ABB RAPID module: P2540SegmentOrg.mod

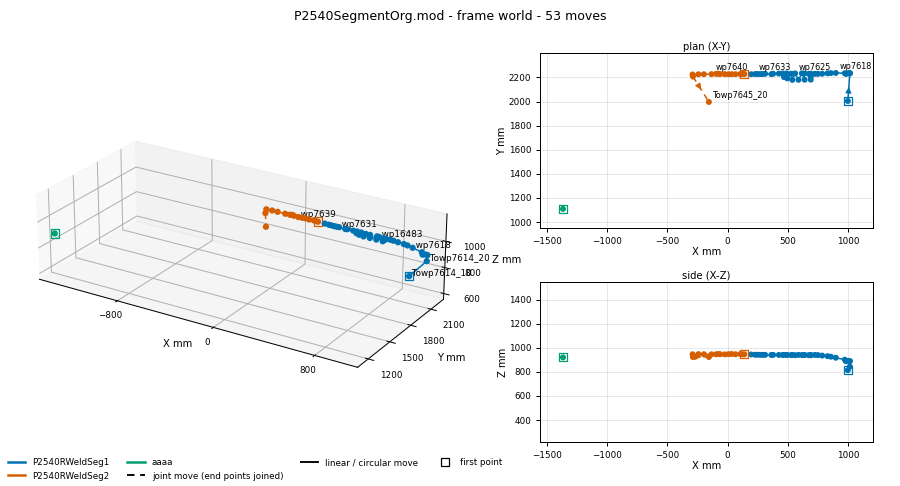
[picture p0: tool path of P2540SegmentOrg.mod in frame world, 53 of 55 moves have a stored position in this frame; points joined in program order, loops and branches not executed]
%%%
   VERSION: 1
   LANGUAGE: ENGLISH
%%%

MODULE P2540Segment
  !********************************
  !*                              *
  !*   Module : P2540Segment.mod   *
  !*   Name   : R1 =2V2=V3AR22    *
  !*   Robot  : 66-60648          *
  !*   Task   : T_Rob1            *
  !*   Vers.  : 7.3               *
  !*                              *
  !********************************
  !
  !
  !============================
  ! Jointtarget for - P2540  -
  !============================
  ! jointtarget for start and stop schedule
  LOCAL CONST jointtarget StartSchedule:=[[23.5621,-44.1357,51.2586,26.8219,73.3194,-96.4131],[9E+09,30.0007,9E+09,9E+09,9E+09,9E+09]];
  LOCAL CONST jointtarget EndSchedule:=[[23.5621,-44.1357,51.2586,26.8219,73.3194,-96.4131],[9E+09,30.0007,9E+09,9E+09,9E+09,9E+09]];
  !
  !
  !===========
  ! Robtarget
  !===========
  ! robtarget for P2540  Right
  LOCAL CONST robtarget Towp7614_10:=[[2081.47,305.36,1121.56],[0.00371606,0.598737,0.800932,-0.000148476],[0,0,-1,0],[9E+09,79.9999,9E+09,9E+09,9E+09,9E+09]];
  LOCAL CONST robtarget Towp7614_20:=[[2062.30,533.66,1090.73],[0.0314135,-0.610941,-0.788905,0.0581832],[0,0,-1,0],[9E+09,59.9996,9E+09,9E+09,9E+09,9E+09]];
  LOCAL CONST robtarget wp7614:=[[2060.79,536.44,1045.07],[0.0756945,-0.590813,-0.799762,0.0747174],[0,0,-1,0],[9E+09,27.201,9E+09,9E+09,9E+09,9E+09]];
  LOCAL CONST robtarget wp7615:=[[2072.79,535.23,1043.37],[0.0761961,-0.650595,-0.752147,0.0720186],[0,0,-1,0],[9E+09,21.5173,9E+09,9E+09,9E+09,9E+09]];
  LOCAL CONST robtarget wp7616:=[[2104.65,535.90,1033.71],[0.0596176,-0.670701,-0.735912,0.0709296],[0,0,-1,0],[9E+09,20.2489,9E+09,9E+09,9E+09,9E+09]];
  LOCAL CONST robtarget wp7619:=[[2219.57,538.20,1009.48],[0.0741953,-0.671905,-0.735684,0.0424222],[0,0,-1,0],[9E+09,27.2002,9E+09,9E+09,9E+09,9E+09]];
  LOCAL CONST robtarget wp7620:=[[2247.39,536.95,1005.37],[0.0595264,-0.701649,-0.708305,0.0494151],[0,0,-1,0],[9E+09,27.2002,9E+09,9E+09,9E+09,9E+09]];
  LOCAL CONST robtarget wp7621:=[[2292.13,533.79,1000.70],[0.0332252,-0.730819,-0.681624,0.013398],[0,0,-1,0],[9E+09,28.1993,9E+09,9E+09,9E+09,9E+09]];
  LOCAL CONST robtarget wp7622:=[[2327.33,533.09,996.92],[0.0333113,-0.730834,-0.681602,0.0134842],[0,0,-1,0],[9E+09,27.2006,9E+09,9E+09,9E+09,9E+09]];
  LOCAL CONST robtarget wp7623:=[[2353.30,533.71,995.86],[0.0293606,-0.749439,-0.661259,0.0143902],[0,0,-1,0],[9E+09,27.1999,9E+09,9E+09,9E+09,9E+09]];
  LOCAL CONST robtarget wp16388:=[[2387.90,486.12,997.86],[0.00612508,-0.760122,-0.649737,-0.00322363],[0,0,-1,0],[9E+09,4.11012,9E+09,9E+09,9E+09,9E+09]];
  LOCAL CONST robtarget wp22643:=[[2386.96,534.93,997.70],[0.0127164,-0.751544,-0.659552,0.00163492],[0,0,-1,0],[9E+09,29.9002,9E+09,9E+09,9E+09,9E+09]];
  LOCAL CONST robtarget wp7624:=[[2405.02,534.99,998.03],[0.000354615,0.772557,0.634784,0.0140377],[0,0,-1,0],[9E+09,29.8997,9E+09,9E+09,9E+09,9E+09]];
  LOCAL CONST robtarget wp16483:=[[2442.71,537.01,996.52],[0.0171293,-0.772749,-0.634461,-0.00402584],[0,0,-1,0],[9E+09,29.9002,9E+09,9E+09,9E+09,9E+09]];
  LOCAL CONST robtarget wp16482:=[[2480.83,537.98,1000.06],[0.000439903,0.773189,0.634169,-0.000630514],[0,0,-1,0],[9E+09,32.3991,9E+09,9E+09,9E+09,9E+09]];
  LOCAL CONST robtarget wp16389:=[[2438.79,486.06,996.71],[0.00848171,-0.773071,-0.634066,-0.0155309],[0,0,-1,0],[9E+09,27.1999,9E+09,9E+09,9E+09,9E+09]];
  LOCAL CONST robtarget wp16390:=[[2489.71,485.99,996.41],[0.0138037,-0.776796,-0.629424,-0.0146608],[0,0,-1,0],[9E+09,4.07069,9E+09,9E+09,9E+09,9E+09]];
  LOCAL CONST robtarget wp7625:=[[2516.82,539.27,998.69],[0.0143354,-0.773193,-0.633743,-0.0181102],[0,0,-1,0],[9E+09,40.9991,9E+09,9E+09,9E+09,9E+09]];
  LOCAL CONST robtarget wp16391:=[[2540.52,486.02,996.53],[0.0108996,-0.789577,-0.613522,-0.00567082],[0,0,-1,0],[9E+09,4.11961,9E+09,9E+09,9E+09,9E+09]];
  LOCAL CONST robtarget wp7626:=[[2549.80,537.47,998.38],[0.00989104,-0.789531,-0.61347,-0.0137525],[0,0,-1,0],[9E+09,32.3999,9E+09,9E+09,9E+09,9E+09]];
  LOCAL CONST robtarget wp16392:=[[2582.12,498.78,997.71],[0.00612506,-0.789608,-0.613429,-0.0133152],[0,0,-1,0],[9E+09,27.3998,9E+09,9E+09,9E+09,9E+09]];
  LOCAL CONST robtarget wp7628:=[[2620.20,540.35,997.67],[0.00660724,0.789817,0.61328,0.00488902],[0,0,-1,0],[9E+09,32.3997,9E+09,9E+09,9E+09,9E+09]];
  LOCAL CONST robtarget wp7630:=[[2652.05,539.44,997.26],[0.00765265,-0.811596,-0.584132,-0.00589266],[0,0,-1,0],[9E+09,32.4003,9E+09,9E+09,9E+09,9E+09]];


  LOCAL CONST robtarget wp16473:=[[2699.16,538.68,997.15],[0.00502678,-0.811529,-0.584197,-0.0100621],[0,0,-1,0],[9E+09,29.9001,9E+09,9E+09,9E+09,9E+09]];
  LOCAL CONST robtarget wp16471:=[[2713.62,536.00,997.85],[0.0220624,-0.810911,-0.584577,-0.0140417],[0,0,-1,0],[9E+09,29.8894,9E+09,9E+09,9E+09,9E+09]];
  LOCAL CONST robtarget wp16472:=[[2727.21,534.57,998.78],[0.000173773,-0.813784,-0.58116,-0.000410488],[0,0,-1,0],[9E+09,31.0445,9E+09,9E+09,9E+09,9E+09]];
  LOCAL CONST robtarget wp7631:=[[2765.83,539.26,997.19],[0.00454817,-0.812585,-0.582806,0.0035711],[0,0,-1,0],[9E+09,29.9004,9E+09,9E+09,9E+09,9E+09]];
  LOCAL CONST robtarget wp31008:=[[2786.44,538.03,997.19],[0.00908552,-0.814655,-0.579848,0.00473351],[0,0,-1,0],[9E+09,29.9001,9E+09,9E+09,9E+09,9E+09]];

  LOCAL CONST robtarget wp7632:=[[2806.45,537.63,997.32],[0.00900133,0.815927,0.578044,0.00628094],[0,0,-1,0],[9E+09,30.0007,9E+09,9E+09,9E+09,9E+09]];
  LOCAL CONST robtarget wp31009:=[[2829.93,538.04,996.73],[0.00768568,0.812719,0.582397,0.0152683],[0,0,-1,0],[9E+09,29.9005,9E+09,9E+09,9E+09,9E+09]];

  LOCAL CONST robtarget wp7633:=[[2848.76,538.17,996.85],[0.00725543,0.810933,0.585076,0.00354437],[0,0,-1,0],[9E+09,29.8994,9E+09,9E+09,9E+09,9E+09]];
  LOCAL CONST robtarget wp7634:=[[2881.59,537.27,994.84],[0.0105951,-0.810906,-0.585073,-0.000189071],[0,0,-1,0],[9E+09,29.9002,9E+09,9E+09,9E+09,9E+09]];
  LOCAL CONST robtarget wp16150:=[[2938.22,539.11,993.71],[0.0155581,-0.812601,-0.582198,-0.0217884],[0,0,-1,0],[9E+09,29.9001,9E+09,9E+09,9E+09,9E+09]];
  LOCAL CONST robtarget wp16151:=[[2973.15,539.53,991.63],[0.0143352,-0.812577,-0.582323,-0.0201075],[0,0,-1,0],[9E+09,29.9001,9E+09,9E+09,9E+09,9E+09]];
  LOCAL CONST robtarget wp7636:=[[3012.11,539.12,993.74],[0.0076257,-0.811727,-0.583768,-0.0157572],[0,0,-1,0],[9E+09,27.2002,9E+09,9E+09,9E+09,9E+09]];
  LOCAL CONST robtarget wp7637:=[[3043.26,539.70,991.91],[0.0186046,-0.811439,-0.583534,-0.0264702],[0,0,-1,0],[9E+09,27.1997,9E+09,9E+09,9E+09,9E+09]];
  LOCAL CONST robtarget wp7638:=[[3070.27,539.54,992.95],[0.00847598,-0.813252,-0.581717,-0.0120917],[0,0,-1,0],[9E+09,27.2002,9E+09,9E+09,9E+09,9E+09]];
  LOCAL CONST robtarget wp7639:=[[3100.66,540.23,995.08],[0.00913472,-0.865282,-0.500928,-0.0163131],[0,0,-1,0],[9E+09,27.2002,9E+09,9E+09,9E+09,9E+09]];
  LOCAL CONST robtarget wp16146:=[[3138.44,541.78,994.19],[0.0055009,-0.894006,-0.447865,-0.0114338],[0,0,-1,0],[9E+09,29.9001,9E+09,9E+09,9E+09,9E+09]];
  LOCAL CONST robtarget wp16411:=[[3156.07,537.38,997.99],[0.00338754,0.895748,0.444538,0.00149798],[0,0,-1,0],[9E+09,60,9E+09,9E+09,9E+09,9E+09]];
  LOCAL CONST robtarget wp16147:=[[3173.12,543.64,994.77],[0.00345947,-0.894048,-0.447902,-0.00641748],[0,0,-1,0],[9E+09,29.9004,9E+09,9E+09,9E+09,9E+09]];
  LOCAL CONST robtarget wp7640:=[[3210.69,541.93,995.09],[0.00726479,-0.896754,-0.442203,-0.0150922],[0,0,-1,0],[9E+09,27.2006,9E+09,9E+09,9E+09,9E+09]];
  LOCAL CONST robtarget wp7642:=[[3274.35,542.16,994.69],[0.00655286,-0.899967,-0.435565,-0.0170478],[0,0,-1,0],[9E+09,27.1997,9E+09,9E+09,9E+09,9E+09]];
  LOCAL CONST robtarget wp7643:=[[3319.94,541.93,994.28],[0.00891136,-0.924508,-0.380439,-0.0215371],[0,0,-1,0],[9E+09,27.2002,9E+09,9E+09,9E+09,9E+09]];
  LOCAL CONST robtarget wp7644:=[[3368.35,541.38,995.77],[0.0101282,-0.928939,-0.369177,-0.0258691],[0,0,-1,0],[9E+09,27.1991,9E+09,9E+09,9E+09,9E+09]];
  LOCAL CONST robtarget Towp7645_20:=[[3235.39,311.48,1018.62],[0.00729107,-0.929368,-0.369063,0.00225485],[0,0,-2,0],[9E+09,58.7207,9E+09,9E+09,9E+09,9E+09]];
  LOCAL CONST robtarget Towp7645_30:=[[3678.48,197.21,1015.08],[0.00379367,0.692205,0.721685,0.000353803],[1,-1,0,0],[9E+09,50,9E+09,9E+09,9E+09,9E+09]];
  LOCAL CONST robtarget wp7645:=[[3426.32,542.43,994.99],[0.0229346,-0.426697,-0.903983,-0.014501],[1,-1,0,0],[9E+09,25,9E+09,9E+09,9E+09,9E+09]];
  LOCAL CONST robtarget wp7647:=[[3515.94,541.61,994.94],[0.0180354,-0.560505,-0.827819,-0.0147185],[1,-1,0,0],[9E+09,20,9E+09,9E+09,9E+09,9E+09]];
  LOCAL CONST robtarget wp7648:=[[3566.36,543.48,994.12],[0.000513143,0.675137,0.737686,-0.000593508],[1,-1,0,0],[9E+09,20,9E+09,9E+09,9E+09,9E+09]];
  LOCAL CONST robtarget wp7649:=[[3616.27,543.9,993.12],[0.000208783,0.783466,0.621428,-0.00029122],[1,0,-1,0],[9E+09,20,9E+09,9E+09,9E+09,9E+09]];

  LOCAL CONST robtarget Frwp6240_20:=[[3468.86,140.72,795.38],[0.00296039,0.761935,0.647638,0.001747],[1,-1,0,0],[9E+09,35.3553,9E+09,9E+09,9E+09,9E+09]];
  !
  !==========
  ! WobjData
  !==========
  ! wobj for spot welding P2540 Right
  PERS wobjdata wP2540_CabFrame:=[FALSE,TRUE,"",[[3089,1731.03,1926.23],[0.00267617,0.00632448,-0.999974,0.00237532]],[[0,0,0],[1,0,0,0]]];
  !
  !
  !==========
  ! SpotData
  !==========
  ! spot data P2540  Right
  LOCAL PERS spotdata Sd_wp7614_30:=[00761430,0,0,0,0];
  LOCAL PERS spotdata Sd_wp7615_30:=[00761530,0,0,0,0];
  LOCAL PERS spotdata Sd_wp7616_30:=[00761630,0,0,0,0];
  LOCAL PERS spotdata Sd_wp7619_30:=[00761930,0,0,0,0];
  LOCAL PERS spotdata Sd_wp7620_30:=[00762030,0,0,0,0];
  LOCAL PERS spotdata Sd_wp7621_30:=[00762130,0,0,0,0];
  LOCAL PERS spotdata Sd_wp7622_30:=[00762230,0,0,0,0];
  LOCAL PERS spotdata Sd_wp7623_30:=[00762330,0,0,0,0];
  LOCAL PERS spotdata Sd_wp7624_30:=[00762430,0,0,0,0];
  LOCAL PERS spotdata Sd_wp16483_30:=[01648330,0,0,0,0];
  LOCAL PERS spotdata Sd_wp16389_30:=[01638930,0,0,0,0];
  LOCAL PERS spotdata Sd_wp16482_30:=[01648230,0,0,0,0];
  LOCAL PERS spotdata Sd_wp16390_30:=[01639030,0,0,0,0];
  LOCAL PERS spotdata Sd_wp7625_30:=[00762530,0,0,0,0];
  LOCAL PERS spotdata Sd_wp16391_30:=[01639130,0,0,0,0];
  LOCAL PERS spotdata Sd_wp7626_30:=[00762630,0,0,0,0];
  LOCAL PERS spotdata Sd_wp16392_30:=[01639230,0,0,0,0];
  LOCAL PERS spotdata Sd_wp7628_30:=[00762830,0,0,0,0];
  LOCAL PERS spotdata Sd_wp7630_30:=[00763030,0,0,0,0];
  LOCAL PERS spotdata Sd_wp16473_30:=[01647330,0,0,0,0];
  LOCAL PERS spotdata Sd_wp16471_30:=[01647130,0,0,0,0];
  LOCAL PERS spotdata Sd_wp16472_30:=[01647230,0,0,0,0];
  LOCAL PERS spotdata Sd_wp7631_30:=[00763130,0,0,0,0];
  LOCAL PERS spotdata Sd_wp31008_30:=[03100830,0,0,0,0];
  LOCAL PERS spotdata Sd_wp31009_30:=[03100930,0,0,0,0];
  LOCAL PERS spotdata Sd_wp7632_30:=[00763230,0,0,0,0];
  LOCAL PERS spotdata Sd_wp7633_30:=[00763330,0,0,0,0];
  LOCAL PERS spotdata Sd_wp7634_30:=[00763430,0,0,0,0];
  LOCAL PERS spotdata Sd_wp16150_30:=[01615030,0,0,0,0];
  LOCAL PERS spotdata Sd_wp16151_30:=[01615130,0,0,0,0];
  LOCAL PERS spotdata Sd_wp7636_30:=[00763630,0,0,0,0];
  LOCAL PERS spotdata Sd_wp7637_30:=[00763730,0,0,0,0];
  LOCAL PERS spotdata Sd_wp7638_30:=[00763830,0,0,0,0];
  LOCAL PERS spotdata Sd_wp7639_30:=[00763930,0,0,0,0];
  LOCAL PERS spotdata Sd_wp16146_30:=[01614630,0,0,0,0];
  LOCAL PERS spotdata Sd_wp16147_30:=[01614730,0,0,0,0];
  LOCAL PERS spotdata Sd_wp7640_30:=[00764030,0,0,0,0];
  LOCAL PERS spotdata Sd_wp7642_30:=[00764230,0,0,0,0];
  LOCAL PERS spotdata Sd_wp7643_30:=[00764330,0,0,0,0];
  LOCAL PERS spotdata Sd_wp7644_30:=[00764430,0,0,0,0];
  LOCAL PERS spotdata Sd_wp7645_30:=[00764530,0,0,0,0];
  LOCAL PERS spotdata Sd_wp7647_30:=[00764730,0,0,0,0];
  LOCAL PERS spotdata Sd_wp7648_30:=[00764830,0,0,0,0];
  LOCAL PERS spotdata Sd_wp22643_30:=[02264330,0,0,0,0];
  LOCAL PERS spotdata Sd_wp16388_30:=[1638830,3880,0,0,0];
  LOCAL PERS spotdata sd_wp16413_30:=[1641330,0,0,0,0];
  LOCAL PERS spotdata Sd_wp34328_30:=[3432830,0,0,0,0];
  LOCAL PERS spotdata sd_wp7617_30:=[761730,0,0,0,0];
  LOCAL PERS spotdata sd_wp7618_30:=[761830,0,0,0,0];
  LOCAL PERS spotdata sd_wp16387_30:=[1638730,0,0,0,0];
  LOCAL PERS spotdata sd_wp16393_30:=[1639330,0,0,0,0];
  LOCAL PERS spotdata sd_wp7627_30:=[762730,0,0,0,0];

  CONST robtarget Towp7645_40:=[[3473.50,534.80,1024.96],[0.00386089,0.504817,0.863213,-0.000495609],[1,-1,0,0],[9E+09,49.9999,9E+09,9E+09,9E+09,9E+09]];
  CONST robtarget Towp7645_10:=[[3365.05,523.37,1018.51],[0.00731169,-0.929363,-0.369076,0.00228623],[0,0,-2,0],[9E+09,58.7205,9E+09,9E+09,9E+09,9E+09]];
  CONST robtarget wp7651:=[[3714.52,543.28,993.87],[0.000278211,0.783469,0.621424,-0.000487569],[1,-1,0,0],[9E+09,27.2004,9E+09,9E+09,9E+09,9E+09]];
  CONST robtarget wp7652:=[[3763.20,543.25,993.02],[0.0003127,0.783489,0.621399,-0.000693894],[1,-1,0,0],[9E+09,27.2,9E+09,9E+09,9E+09,9E+09]];
  CONST robtarget wp6240:=[[3909.48,543.88,995.46],[0.000317241,0.784542,0.620068,-0.000736588],[1,-1,0,0],[9E+09,27.2012,9E+09,9E+09,9E+09,9E+09]];
  CONST robtarget Towp6240_10:=[[3908.13,534.59,1007.05],[0.000276509,-0.78458,-0.620021,-0.000767366],[1,-1,0,0],[9E+09,40,9E+09,9E+09,9E+09,9E+09]];
  CONST robtarget Frwp6240_10:=[[3605.82,222.30,1026.08],[0.000211859,0.691607,0.722259,0.00360361],[1,-1,0,0],[9E+09,51.511,9E+09,9E+09,9E+09,9E+09]];
  CONST robtarget Frwp6240_30:=[[3423.48,113.69,718.92],[0.00387007,0.783505,0.621365,0.00112283],[1,0,-1,0],[9E+09,30.0015,9E+09,9E+09,9E+09,9E+09]];
  LOCAL CONST robtarget wp34328:=[[3154.52,544.41,992.22],[0.00232207,-0.894068,-0.44789,-0.00477992],[0,0,-1,0],[9E+09,29.9001,9E+09,9E+09,9E+09,9E+09]];
  CONST robtarget wp7646:=[[2138.86,539.12,1028.14],[0.0666694,-0.672846,-0.734889,0.0525741],[0,0,-1,0],[9E+09,26.3985,9E+09,9E+09,9E+09,9E+09]];
  CONST robtarget wp7617:=[[2138.85,539.12,1028.13],[0.0666662,-0.672844,-0.73489,0.0525757],[0,0,-1,0],[9E+09,26.3981,9E+09,9E+09,9E+09,9E+09]];
  CONST robtarget wp7127:=[[2178.03,541.13,1019.79],[0.0665654,-0.672821,-0.734926,0.0524885],[0,0,-1,0],[9E+09,26.3969,9E+09,9E+09,9E+09,9E+09]];
  CONST robtarget wp7618:=[[2179.08,538.86,1017.92],[0.0760443,-0.671726,-0.73419,0.0629157],[0,0,-1,0],[9E+09,19.3525,9E+09,9E+09,9E+09,9E+09]];
  CONST robtarget wp22653:=[[2387.26,520.57,998.85],[0.000174384,0.753397,0.65756,-0.00010412],[0,0,-1,0],[9E+09,32.3975,9E+09,9E+09,9E+09,9E+09]];
  CONST robtarget wp16387:=[[2387.15,512.63,997.92],[0.0104316,-0.753264,-0.657466,-0.0146614],[0,0,-1,0],[9E+09,4.91916,9E+09,9E+09,9E+09,9E+09]];
  CONST robtarget wp16402:=[[2609.28,509.65,999.16],[0.00365543,0.789724,0.613444,0.000838796],[0,0,-1,0],[9E+09,27.3982,9E+09,9E+09,9E+09,9E+09]];
  CONST robtarget wp16393:=[[2609.30,509.71,996.41],[0.00424136,-0.789644,-0.613445,-0.0110424],[0,0,-1,0],[9E+09,27.2006,9E+09,9E+09,9E+09,9E+09]];
  CONST robtarget wp16403:=[[2583.99,537.89,999.25],[0.00370574,0.789724,0.613444,0.000907163],[0,0,-1,0],[9E+09,27.3972,9E+09,9E+09,9E+09,9E+09]];
  CONST robtarget wp7627:=[[2587.97,540.22,997.14],[0.0035651,-0.789261,-0.614038,-0.00196816],[0,0,-1,0],[9E+09,32.4011,9E+09,9E+09,9E+09,9E+09]];
  CONST robtarget wp16160:=[[2954.69,538.15,995.29],[0.00375398,0.813115,0.582082,0.00111285],[0,0,-1,0],[9E+09,32.4004,9E+09,9E+09,9E+09,9E+09]];
  CONST robtarget wp16413:=[[2954.96,539.94,993.87],[0.0162414,-0.812446,-0.582331,-0.0234421],[0,0,-1,0],[9E+09,29.9004,9E+09,9E+09,9E+09,9E+09]];
  CONST robtarget wp16399:=[[2460.90,539.36,1000.13],[0.000463969,0.773187,0.634171,-0.000603479],[0,0,-1,0],[9E+09,32.4005,9E+09,9E+09,9E+09,9E+09]];
  LOCAL CONST robtarget wp16481:=[[2460.82,539.63,997.22],[0.014924,-0.773008,-0.63421,-0.00227041],[0,0,-1,0],[9E+09,29.9005,9E+09,9E+09,9E+09,9E+09]];
  LOCAL PERS spotdata Sd_wp16481_30:=[1648130,0,0,0,0];
  CONST robtarget wp7635:=[[2094.70,529.51,1046.98],[0.0624239,-0.652073,-0.753492,0.0560746],[0,0,-1,0],[9E+09,27.1997,9E+09,9E+09,9E+09,9E+09]];
  LOCAL PERS spotdata Sd_wp425935:=[1615130,0,0,0,0];
  !
  !
  !
  !
  !
  !-------------------------
  ! Spot Welding P2540  Right
  !-------------------------
  PROC P2540RWeldSeg1()
    ! Rob1 - P2540 Right -
    ToolLoad XQ11GunTCP,loXQ11Gun;
    !curr_simdata.sim_type := 0;
    MoveAbsJ StartSchedule,v200,fine,XQ11GunTCP;
    MoveJ Towp7614_10,v2500,z80,XQ11GunTCP\WObj:=wP2540_CabFrame;
    MoveL Towp7614_20,v2500,z80,XQ11GunTCP\WObj:=wP2540_CabFrame;
    SpotL wp7614,v2500,XQ11Gun,Sd_wp7614_30,XQ11GunTCP\WObj:=wP2540_CabFrame;
    SpotL wp7615,v2500,XQ11Gun,Sd_wp7615_30,XQ11GunTCP\WObj:=wP2540_CabFrame;
    MoveL wp7635, v2500, z80, XQ11GunTCP\WObj:=wP2540_CabFrame;
    SpotL wp7616,v2500,XQ11Gun,Sd_wp7616_30,XQ11GunTCP\WObj:=wP2540_CabFrame;
    SpotL wp7618, v2500, XQ11Gun, sd_wp7618_30, XQ11GunTCP\WObj:=wP2540_CabFrame;
    SpotL wp7619,v2500,XQ11Gun,Sd_wp7619_30,XQ11GunTCP\WObj:=wP2540_CabFrame;
    SpotL wp7620,v2500,XQ11Gun,Sd_wp7620_30,XQ11GunTCP\WObj:=wP2540_CabFrame;
    SpotL wp7621,v2500,XQ11Gun,Sd_wp7621_30,XQ11GunTCP\WObj:=wP2540_CabFrame;
    SpotL wp7622,v2500,XQ11Gun,Sd_wp7622_30,XQ11GunTCP\WObj:=wP2540_CabFrame;
    SpotL wp7623,v2500,XQ11Gun,Sd_wp7623_30,XQ11GunTCP\WObj:=wP2540_CabFrame;
    SpotL wp22643,v2500,XQ11Gun,Sd_wp22643_30,XQ11GunTCP\WObj:=wP2540_CabFrame;
    SpotL wp16387, v2500, XQ11Gun, sd_wp16387_30, XQ11GunTCP\WObj:=wP2540_CabFrame;
    SpotL wp16388,v2500,XQ11Gun,Sd_wp16388_30,XQ11GunTCP\WObj:=wP2540_CabFrame;
    SpotL wp7624,v2500,XQ11Gun,Sd_wp7624_30,XQ11GunTCP\WObj:=wP2540_CabFrame;
    SpotL wp16483,v2500,XQ11Gun,Sd_wp16483_30,XQ11GunTCP\WObj:=wP2540_CabFrame;
    SpotL wp16389,v2500,XQ11Gun,Sd_wp16389_30,XQ11GunTCP\WObj:=wP2540_CabFrame;
    SpotL wp16481, v2500, XQ11Gun, Sd_wp16481_30, XQ11GunTCP\WObj:=wP2540_CabFrame;
    SpotL wp16390,v2500,XQ11Gun,Sd_wp16390_30,XQ11GunTCP\WObj:=wP2540_CabFrame;
    SpotL wp7625,v2500,XQ11Gun,Sd_wp7625_30,XQ11GunTCP\WObj:=wP2540_CabFrame;
    SpotL wp16391,v2500,XQ11Gun,Sd_wp16391_30,XQ11GunTCP\WObj:=wP2540_CabFrame;
    SpotL wp7626,v2500,XQ11Gun,Sd_wp7626_30,XQ11GunTCP\WObj:=wP2540_CabFrame;
    SpotL wp16392,v2500,XQ11Gun,Sd_wp16392_30,XQ11GunTCP\WObj:=wP2540_CabFrame;
    SpotL wp16393, v2500, XQ11Gun, sd_wp16393_30, XQ11GunTCP\WObj:=wP2540_CabFrame;
    SpotL wp7627, v2500, XQ11Gun, sd_wp7627_30, XQ11GunTCP\WObj:=wP2540_CabFrame;
    SpotL wp7628,v2500,XQ11Gun,Sd_wp7628_30,XQ11GunTCP\WObj:=wP2540_CabFrame;
    SpotL wp7630,v2500,XQ11Gun,Sd_wp7630_30,XQ11GunTCP\WObj:=wP2540_CabFrame;
    SpotL wp16473,v2500,XQ11Gun,Sd_wp16473_30,XQ11GunTCP\WObj:=wP2540_CabFrame;
    SpotL wp16471,v2500,XQ11Gun,Sd_wp16471_30,XQ11GunTCP\WObj:=wP2540_CabFrame;
    !SpotL wp16472,v2500,XQ11Gun,Sd_wp16472_30,XQ11GunTCP\WObj:=wP2540_CabFrame;
    SpotL wp7631,v2500,XQ11Gun,Sd_wp7631_30,XQ11GunTCP\WObj:=wP2540_CabFrame;
    ! 31008
    SpotL wp31008, v2500, XQ11Gun, Sd_wp31008_30, XQ11GunTCP\WObj:=wP2540_CabFrame;
    SpotL wp7632,v2500,XQ11Gun,Sd_wp7632_30,XQ11GunTCP\WObj:=wP2540_CabFrame;
    ! 31009
    SpotL wp31009, v2500, XQ11Gun, Sd_wp31009_30, XQ11GunTCP\WObj:=wP2540_CabFrame;
    SpotL wp7633,v2500,XQ11Gun,Sd_wp7633_30,XQ11GunTCP\WObj:=wP2540_CabFrame;
    SpotL wp7634,v2500,XQ11Gun,Sd_wp7634_30,XQ11GunTCP\WObj:=wP2540_CabFrame;

    ! end
  ENDPROC

  !----------
  PROC P2540RWeldSeg2()
    SpotL wp16150,v2500,XQ11Gun,Sd_wp16150_30,XQ11GunTCP\WObj:=wP2540_CabFrame;
    SpotL wp16413, v2500, XQ11Gun, sd_wp16413_30, XQ11GunTCP\WObj:=wP2540_CabFrame;
    SpotL wp16151,v2500,XQ11Gun,Sd_wp16151_30,XQ11GunTCP\WObj:=wP2540_CabFrame;
    !
    SpotL wp7636,v2500,XQ11Gun,Sd_wp7636_30,XQ11GunTCP\WObj:=wP2540_CabFrame;
    SpotL wp7637,v2500,XQ11Gun,Sd_wp7637_30,XQ11GunTCP\WObj:=wP2540_CabFrame;
    SpotL wp7638,v2500,XQ11Gun,Sd_wp7638_30,XQ11GunTCP\WObj:=wP2540_CabFrame;
    SpotL wp7639,v2500,XQ11Gun,Sd_wp7639_30,XQ11GunTCP\WObj:=wP2540_CabFrame;
    !
    SpotL wp16146,v2500,XQ11Gun,Sd_wp16146_30,XQ11GunTCP\WObj:=wP2540_CabFrame;
    SpotL wp34328, v2500, XQ11Gun, Sd_wp34328_30, XQ11GunTCP\WObj:=wP2540_CabFrame;
    SpotL wp16147,v2500,XQ11Gun,Sd_wp16147_30,XQ11GunTCP\WObj:=wP2540_CabFrame;
    SpotL wp7640,v2500,XQ11Gun,Sd_wp7640_30,XQ11GunTCP\WObj:=wP2540_CabFrame;
    SpotL wp7642,v2500,XQ11Gun,Sd_wp7642_30,XQ11GunTCP\WObj:=wP2540_CabFrame;
    SpotL wp7643,v2500,XQ11Gun,Sd_wp7643_30,XQ11GunTCP\WObj:=wP2540_CabFrame;
    SpotL wp7644,v2500,XQ11Gun,Sd_wp7644_30,XQ11GunTCP\WObj:=wP2540_CabFrame;
    MoveL Towp7645_10, v1000, z50, XQ11GunTCP\WObj:=wP2540_CabFrame;
    MoveJ Towp7645_20,v2500,z80,XQ11GunTCP\WObj:=wP2540_CabFrame;
  ENDPROC

  !----------
  PROC P2540RWeldSeg3()
    ! Rob1 - P2540 Right -
    ToolLoad XQ11GunTCP,loXQ11Gun;
    !MoveJ Towp7645_30,v2500,z80,XQ11GunTCP\WObj:=wP2540_CabFrame;
    !MoveL Towp7645_40, v2500, z80, XQ11GunTCP\WObj:=wP2540_CabFrame;
    !SpotL wp7645,v2500,XQ11Gun,Sd_wp7645_30,XQ11GunTCP\WObj:=wP2540_CabFrame;
    !SpotL wp7647,v2500,XQ11Gun,Sd_wp7647_30,XQ11GunTCP\WObj:=wP2540_CabFrame;
    !SpotL wp7648,v2500,XQ11Gun,Sd_wp7648_30,XQ11GunTCP\WObj:=wP2540_CabFrame;


    ! end
  ENDPROC

  !----------

  PROC P2540RWeldSeg4()
    ! Rob1 - P2540 Left -
    ToolLoad XQ11GunTCP,loXQ11Gun;
    !MoveL Frwp6240_10, v1000, z50, XQ11GunTCP\WObj:=wP2540_CabFrame;
    !MoveL Frwp6240_20,v2500,z80,XQ11GunTCP\WObj:=wP2540_CabFrame;
    !MoveL Frwp6240_30, v2500, z80, XQ11GunTCP\WObj:=wP2540_CabFrame;
    WeldGunData{1}    .release_dist := 15;
    MoveAbsJ EndSchedule,v2500,fine,XQ11GunTCP;
    !curr_simdata.sim_type := 2;
    ! end
  ENDPROC
  !----------

  !===============
  ! End Of Module
  !===============
	PROC aaaa()
		SpotL [[-1366.65,1108.96,920.06],[0.00444309,-0.038809,-0.00344693,0.999226],[1,0,-2,0],[9E+09,115.501,9E+09,9E+09,9E+09,9E+09]], vmax, XQ11Gun, Sd_wp7614_30, XQ11GunTCP;
	ENDPROC
ENDMODULE
